// TIA Portal V19 export
DATA_BLOCK "MODE SELECTION"   // DB27
{ S7_Optimized_Access := 'FALSE' }
   VAR
      AUTO : Bool;
      MANUAL : Bool;
      STANDBY : Bool;
      "MODE BUFFER" : Int;
   END_VAR
BEGIN
END_DATA_BLOCK
